FUNCTION_BLOCK FB_Bereichsueberwachung
VAR_INPUT
	/// Sollwert 
	in_sollwert: REAL;
	/// Istwert 
	in_istwert: REAL;
	/// Offset Obergrenze 
	in_offset_oben: REAL;
	/// Offset Untergrenze 
	in_offset_unten: REAL;
	/// Freigabe zum Überwachen 
	in_freigabe: BOOL;
END_VAR
VAR_OUTPUT
	/// Sollwerrt im Bereichsfenster (Sollwert= Istwert +/- Offset) 
	out_im_bereich: BOOL;
END_VAR
VAR
	temp_oben_real: REAL;
	temp_unten_real: REAL;
	temp_grenze_oben: BOOL;
	temp_grenze_unten: BOOL;
END_VAR

	(* Obergrenze überschritten ? *)
	temp_oben_real := in_sollwert +in_offset_oben;
	temp_grenze_oben := in_istwert > temp_oben_real;

	(* Untergrenze unterschritten ? *)
	temp_unten_real := in_sollwert - in_offset_unten;
	temp_grenze_unten := in_istwert < temp_unten_real;

	(* Wert liegt im zulässigen Bereich *)
	out_im_bereich := in_freigabe
					AND NOT temp_grenze_unten
					AND NOT temp_grenze_oben;

END_FUNCTION_BLOCK

(* stored: Version 1.1.0.1
   POU FB_Bereichsueberwachung: Id {54f2f6da-64c0-443e-8e32-e71a05c88b4e}, SpecialFunc None *)
